{attribute 'linkalways'} 
{attribute 'no_explicit_call' := 'This FB is a CLASS and must be accessed using methods or properties'}
{attribute 'enable_dynamic_creation'}
FUNCTION_BLOCK Node_F_VN_DrawLines EXTENDS VisionNode
VAR
    ipLines : _ITcVnContainer;
    nLineIndex : _DINT(0);
    ipDestImage : _ITcVnImage;
    aColor : _TcVnVector4_LREAL;
    nThickness : _DINT(1);
    hrPrev : _HRESULT(S_OK);
	hresult : _HRESULT(S_OK);
END_VAR

METHOD PUBLIC  Clone : I_Node
VAR
	pNode : POINTER TO Node_F_VN_DrawLines;
END_VAR
pNode := __NEW(Node_F_VN_DrawLines);
Clone := pNode^;
END_METHOD

METHOD FB_init : BOOL
VAR_INPUT
	bInitRetains : BOOL; // if TRUE, the retain variables are initialized (warm start / cold start)
	bInCopyCode : BOOL;  // if TRUE, the instance afterwards gets moved into the copy code (online change)
END_VAR
AddInput('ipLines', ipLines);
AddParameter('nLineIndex', nLineIndex);
AddInput('ipDestImage', ipDestImage);
AddInput('aColor', aColor);
AddParameter('nThickness', nThickness);
AddInput('hrPrev', hrPrev);
AddOutput('ipDestImage', ipDestImage);
AddOutput('hresult',hresult);
END_METHOD

METHOD PROTECTED OnExecute
hresult.Value := F_VN_DrawLines(
    ipLines := ipLines.Value,
    nLineIndex := nLineIndex.Value,
	ipDestImage := ipDestImage.Value,
    aColor := aColor.Value,
    nThickness := nThickness.Value,
	hrPrev:= hrPrev.Value);
END_METHOD

METHOD PUBLIC PreExecutionCheck
VAR_INPUT
	Check : I_PreExecutionChecks;
END_VAR
Check.IsTrue(ipLines.IsValid, 'ipLines must be a valid container');

Check.IsTrue((ipLines.IsType(TC_GLOBAL_CONST_LIST.ContainerType_Vector_TcVnVector2_REAL) OR
              ipLines.IsType(TC_GLOBAL_CONST_LIST.ContainerType_Vector_TcVnVector4_LREAL) OR
              ipLines.IsType(TC_GLOBAL_CONST_LIST.ContainerType_Vector_TcVnVector4_DINT)),
              'ipLines contains incorrect type');
              
Check.IsTrue(ipDestImage.IsValid, 'ipDestImage must contain an image');
Check.IsTrue(nThickness.Value >= 1, 'nThickness must be greater than or equal to 1');
END_METHOD

END_FUNCTION_BLOCK

(* stored: Version 1.1.0.1, ProductVersion 3.1.4026.13
   POU Node_F_VN_DrawLines: Id {c817b75d-e070-0d56-1723-97be2e3432b3}, SpecialFunc None
   Folder Constructor: Id {77f4399a-c80c-00ba-3739-8b642ff15c04}
   Method Clone: Id {9ac89637-e732-0ba2-0c9e-c24e4480334d}
   Method FB_init: Id {bcee5488-7992-0f86-1329-8509c03d55f0}
   Method OnExecute: Id {ad504b70-737b-0aa2-2989-016ad0304d7f}
   Method PreExecutionCheck: Id {2ef2ea0f-9823-013d-32b9-85b4908b23dd} *)
